FUNCTION BytesToIpv4 : T_IPv4Addr
VAR_INPUT
    IpAddress : ARRAY [0..3] OF BYTE;
END_VAR
VAR
	TempStr	: STRING;
END_VAR


TempStr := CONCAT(TempStr, BYTE_TO_STRING(IpAddress[3]));

TempStr := CONCAT(TempStr, '.');

TempStr := CONCAT(TempStr, BYTE_TO_STRING(IpAddress[2]));

TempStr := CONCAT(TempStr, '.');

TempStr := CONCAT(TempStr, BYTE_TO_STRING(IpAddress[1]));

TempStr := CONCAT(TempStr, '.');

TempStr := CONCAT(TempStr, BYTE_TO_STRING(IpAddress[0]));

BytesToIpv4 := TempStr;

RETURN;

END_FUNCTION

(* stored: Version 1.1.0.1
   POU BytesToIpv4: Id {8ecba468-c83a-4490-8186-c443d9214b5a}, SpecialFunc None *)
